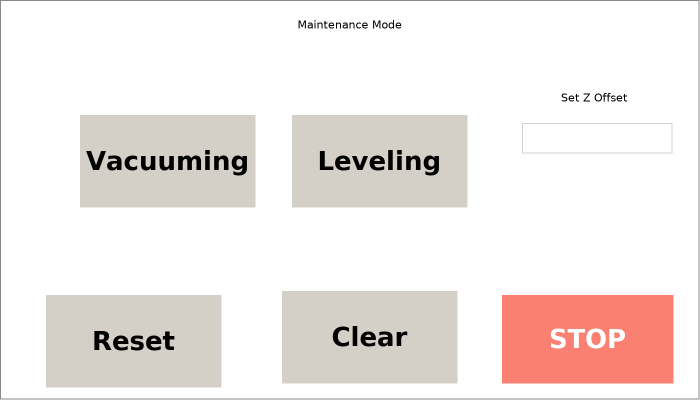
VISUALIZATION V_MaintenanceMode  // 700x400
VAR_IN_OUT
	HMI : ST_PackMLBaseModule_HMI;
END_VAR
    Label (0,0 700x50), "Maintenance Mode"
    RoundedRectangle (282,291 175x92), "Clear"
        OnMouseClick: execute { HMI.Command.State := E_PMLCommand.ePMLCommand_Clear; }
    RoundedRectangle (46,295 175x92), "Reset"
        OnMouseClick: execute { HMI.Command.State := E_PMLCommand.ePMLCommand_Reset; }
    RoundedRectangle (500,293 175x92), "STOP"
        toggle GVL_Safety.eStopHMI
        OnMouseClick: execute {  }
    RoundedRectangle (80,115 175x92), "Vacuuming"
        OnMouseClick: execute { HMI.Command.State := E_PMLCommand.ePMLCommand_Reset; }
    RoundedRectangle (292,115 175x92), "Leveling"
        OnMouseClick: execute { HMI.Command.State := E_PMLCommand.ePMLCommand_Reset; }
    Textfield (522,123 150x30)
    Label (534,83 121x30), "Set Z Offset"
END_VISUALIZATION

(* stored: Version 1.1.0.1, ProductVersion 3.1.4024.15
   Visu V_MaintenanceMode: Id {beddd7b9-7d38-4b95-a44e-95ac60c56cdb} *)
